{attribute 'no_explicit_call' := 'direct call for this function block is not allowed'}
FUNCTION_BLOCK FINAL FB_EmptyWithImplRPC
IMPLEMENTS I_WithRPC
VAR
END_VAR

// A method with all types of input and outputs as well as a return type.
{attribute 'TcRpcEnable'}
METHOD FullMethod : UDINT
VAR_INPUT
	InArg1  	: STRING(64);
	InArg2		: Tc2_System.ST_CpuCoreInfo; 
END_VAR
VAR_IN_OUT
	InOutArg1	: POINTER TO __UXINT;
END_VAR
VAR_OUTPUT
	OutArg1		: Tc2_System.E_SeekOrigin;
	OutArg2		: Tc2_System.T_MaxString;
END_VAR
END_METHOD

// First property.
{attribute 'TcRpcEnable'}
PROPERTY Prop1 : BOOL
GET
END_GET
SET
END_SET
END_PROPERTY

// A method that has no arguments.
{attribute 'TcRpcEnable'}
METHOD VoidMethod
VAR_INPUT
END_VAR
END_METHOD

END_FUNCTION_BLOCK

(* stored: Version 1.1.0.1, ProductVersion 3.1.4024.15
   POU FB_EmptyWithImplRPC: Id {79c30132-5eef-47f4-b006-5599731dc524}, SpecialFunc None
   Method FullMethod: Id {62458351-a809-4bc8-a012-d482669530a0}
   Property Prop1: Id {736d1615-1bcd-4628-99c3-7c6dbe81338d}
   Get Get: Id {6660328d-863a-454c-a315-18eca600c6b8}
   Set Set: Id {87ee97cf-fae3-4766-b9df-cba583e1a2fa}
   Method VoidMethod: Id {5089172c-8c37-45c0-806f-614ab22dceeb} *)
